(* PLC project  *)

PROGRAM P
  VAR
    tmr : TON;
  END_VAR

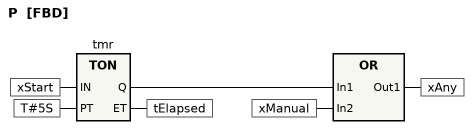
(* FBD diagram, written out as Structured Text *)
tmr(IN := xStart, PT := T#5S);
tElapsed := tmr.ET;
xAny := tmr.Q OR xManual;
END_PROGRAM
